// TwinCAT 3 PLC project MainPlc
// ProgramVersion: 3.1.4023.0
// libraries:
//   Tc2_Standard, * (Beckhoff Automation GmbH)
//   Tc2_System, * (Beckhoff Automation GmbH)
//   Tc3_Module, * (Beckhoff Automation GmbH)
// project tree:
//   / PlcTask.TcTTO (not stored)
//   POUs/ fbPneumaticActuator.TcPOU, MAIN.TcPOU

// ---- POUs/fbPneumaticActuator.TcPOU
FUNCTION_BLOCK fbPneumaticActuator
VAR_INPUT
inRetracted : BOOL;
inExtended : BOOL;
END_VAR
VAR_OUTPUT
	outRetract : BOOL;
	outExtend : BOOL;
END_VAR
VAR
	_manualRetract : BOOL;
	_manualExtend : BOOL;
	_simulatedPosition : INT;
END_VAR

METHOD Extend : BOOL
VAR_INPUT
END_VAR
THIS^.outRetract := FALSE;
THIS^.outExtend := TRUE;

Extend := THIS^.inExtended;
END_METHOD

METHOD Manual : BOOL
VAR_INPUT
END_VAR
IF(THIS^._manualExtend AND_THEN THIS^.Extend()) THEN THIS^._manualExtend := FALSE; END_IF;
IF(THIS^._manualRetract AND_THEN THIS^.Retract()) THEN THIS^._manualRetract := FALSE; END_IF;

THIS^._manualExtend := FALSE;
THIS^._manualRetract := FALSE;
END_METHOD

METHOD Retract : BOOL
VAR_INPUT
END_VAR
THIS^.outRetract := TRUE;
THIS^.outExtend := FALSE;

Retract := THIS^.inRetracted;
END_METHOD

METHOD SimulateInputs : BOOL
VAR_INPUT
END_VAR
IF THIS^.outExtend THEN
	THIS^.inRetracted := FALSE;
	_simulatedPosition := _simulatedPosition + 1;
	IF _simulatedPosition >= 100 THEN
		_simulatedPosition := 100;
		THIS^.inExtended := TRUE;
	END_IF
END_IF
IF outRetract THEN
	THIS^.inExtended := FALSE;
	_simulatedPosition := _simulatedPosition - 1;
	IF _simulatedPosition <= -100 THEN
		_simulatedPosition := -100;
		THIS^.inRetracted := TRUE;
	END_IF
END_IF
END_METHOD

END_FUNCTION_BLOCK

// ---- POUs/MAIN.TcPOU
PROGRAM MAIN
VAR
	_fbPneumaticActuator : fbPneumaticActuator;
END_VAR

_fbPneumaticActuator.Manual();
_fbPneumaticActuator.SimulateInputs();

END_PROGRAM
